# EPICS autosave request: soft_iocs/18id_con/18id/iocBoot/ioc18id/auto_settings.req
file "LabJack_T4_settings.req", P=$(P), N=1
file built_settings.req P=$(P)
